FUNCTION_BLOCK F_LE (* less or equal *)
  (* Standard: 61131-3; Classification: standard comparison function; Description: Copyright (c) 2013 TU Wien ACIN This program and the accompanying materials are made available under the terms of the Eclipse Public License 2.0 which is available at https://www.eclipse.org/legal/epl-2.0/ SPDX-License-Identifier: EPL-2.0 *)
  (* Version 1.0, 2013-03-13, Monika Wenger, TU Wien ACIN *)
  (* Version 3.0, 2025-04-14, Patrick Aigner, changed package *)
  PACKAGE iec61131::comparison;
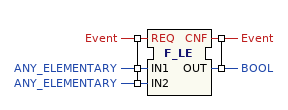
  EVENT_INPUT
    REQ WITH IN1, IN2; (* Service Request *)
  END_EVENT
  EVENT_OUTPUT
    CNF WITH OUT; (* Confirmation of Requested Service *)
  END_EVENT
  VAR_INPUT
    IN1 : ANY_ELEMENTARY; (* Input value 1 *)
    IN2 : ANY_ELEMENTARY; (* Input value 2 *)
  END_VAR
  VAR_OUTPUT
    OUT : BOOL; (* value 1 <= value2 = true *)
  END_VAR
END_FUNCTION_BLOCK
